KUKA KRL program: OTW_CHWYTAK.src

&ACCESS RVO1
&REL 4
&PARAM TEMPLATE = C:\KRC\Roboter\Template\vorgabe
&PARAM EDITMASK = *
DEF OTW_CHWYTAK( )
;FOLD INI
  ;FOLD BASISTECH INI
    GLOBAL INTERRUPT DECL 3 WHEN $STOPMESS==TRUE DO IR_STOPM ( )
    INTERRUPT ON 3
    BAS (#INITMOV,0 )
  ;ENDFOLD (BASISTECH INI)
  ;FOLD USER INI
    ;Make your modifications here

  ;ENDFOLD (USER INI)
;ENDFOLD (INI)

$OUT[5] = FALSE
PULSE($OUT[6],TRUE,0.9)
$OUT[7] = TRUE
WAIT FOR $OUT[6] == FALSE
$OUT[7] = FALSE

END
